# EPICS substitutions: iocBoot/ioc4idVCDM/substitutions/fb_epid.substitutions
# $Id$

file "$(OPTICS)/opticsApp/Db/fb_epid.db"
  {
    {
        P=4idVCDM:epid1,
	IN=4idVCDM:epid1:sim.VAL,
	OUT=4idVCDM:epid1:sim.D,
	MODE=PID,
	CALC=A,
	PERMIT1="4idVCDM:epid1:on.VAL",
	PERMIT2="",
	PERMIT3="",
	PERMIT4=""
    }
  }
